{attribute 'no_explicit_call' := 'do not call this function block directly'}
FUNCTION_BLOCK FB_Vector IMPLEMENTS I_Vector, I_Addition, I_Subtraction, I_Multiplication
VAR
	_fX, _fY, _fZ : LREAL;
END_VAR

{attribute 'hide'}
METHOD FB_init : BOOL
VAR_INPUT
	bInitRetains : BOOL; // if TRUE, the retain variables are initialized (warm start / cold start)
	bInCopyCode : BOOL;  // if TRUE, the instance afterwards gets moved into the copy code (online change)
	fX, fY, fZ : LREAL;
END_VAR
THIS^.SetValue(fX, fY, fZ);
END_METHOD

METHOD Minus : I_Subtraction
VAR_INPUT
	ipObject : I_Object;
END_VAR
VAR_OUTPUT
	e : E_OperatorError;
END_VAR
VAR
	ipVector : I_Vector;
END_VAR
Minus := THIS^;

IF NOT __QUERYINTERFACE(ipObject, ipVector) THEN
  e := E_OperatorError.TypeMismatch;
  RETURN;
  END_IF

THIS^._fX := THIS^._fX - ipVector.X;
THIS^._fY := THIS^._fY - ipVector.Y;
THIS^._fZ := THIS^._fZ - ipVector.Z;
END_METHOD

METHOD Plus : I_Addition
VAR_INPUT
	ipObject : I_Object;
END_VAR
VAR_OUTPUT
	e : E_OperatorError;
END_VAR
VAR
	ipVector : I_Vector;
END_VAR
Plus := THIS^;

IF NOT __QUERYINTERFACE(ipObject, ipVector) THEN
  e := E_OperatorError.TypeMismatch; 
  RETURN;
  END_IF

THIS^._fX := THIS^._fX + ipVector.X;
THIS^._fY := THIS^._fY + ipVector.Y;
THIS^._fZ := THIS^._fZ + ipVector.Z;
END_METHOD

METHOD SetValue : REFERENCE TO FB_Vector
VAR_INPUT
	fX, fY, fZ : LREAL;
END_VAR
SetValue REF= THIS^;

THIS^._fX := fX;
THIS^._fY := fY;
THIS^._fZ := fZ;
END_METHOD

METHOD Times : I_Multiplication
VAR_INPUT
	ipObject : I_Object;
END_VAR
VAR_OUTPUT
	e : E_OperatorError;
END_VAR
VAR
	ipNumber : I_Scalar;
	ipVector : I_Vector;
	TmpX, TmpY, TmpZ : LREAL;
END_VAR
Times := THIS^;

// Scale vector.
IF __QUERYINTERFACE(ipObject, ipNumber) THEN 
	THIS^.SetValue( THIS^._fX * ipNumber.ToF64(),
					THIS^._fY * ipNumber.ToF64(),
					THIS^._fZ * ipNumber.ToF64());
	RETURN;
	END_IF

// Do the cross-product.
IF __QUERYINTERFACE(ipObject, ipVector) THEN 
	TmpX := THIS^._fX;
  TmpY := THIS^._fY;
  TmpZ := THIS^._fZ;
  
	THIS^.SetValue(	(TmpY*ipVector.Z) - (TmpZ*ipVector.Y),
					        (TmpZ*ipVector.X) - (TmpX*ipVector.Y),
					        (TmpX*ipVector.Y) - (TmpY*ipVector.X));
	
	RETURN; 
	END_IF

e := E_OperatorError.TypeMismatch;
END_METHOD

METHOD ToArray : ARRAY[0..2] OF LREAL
VAR_INPUT
END_VAR

ToArray[0]:= THIS^._fX;
ToArray[1]:= THIS^._fY;
ToArray[2]:= THIS^._fZ;
END_METHOD

PROPERTY X : LREAL
GET
X := THIS^._fX;
END_GET
SET
THIS^._fX := X;
END_SET
END_PROPERTY

PROPERTY Y : LREAL
GET
Y := THIS^._fY;
END_GET
SET
THIS^._fY:= Y;
END_SET
END_PROPERTY

PROPERTY Z : LREAL
GET
Z := THIS^._fZ;
END_GET
SET
THIS^._fZ := Z;
END_SET
END_PROPERTY

END_FUNCTION_BLOCK

(* stored: Version 1.1.0.1, ProductVersion 3.1.4024.12
   POU FB_Vector: Id {a3e3f989-5383-4684-9365-351b5d5ddbc2}, SpecialFunc None
   Folder Constructor: Id {4d519fb7-d67d-4a3b-ad25-276b7aa36544}
   Folder IOperatorX: Id {dc5b5d9f-5cca-45c6-8635-d968a0da61ca}
   Folder IVector: Id {a72ffef8-55b1-4923-ae3f-21af8125f718}
   Method FB_init: Id {5e146931-1a8b-485c-a8f5-25b63288d0d0}
   Method Minus: Id {8d6c7050-0ff6-4ab0-a242-534401decfff}
   Method Plus: Id {5087b5ff-4e99-4c43-993f-4b57fa3ce74e}
   Method SetValue: Id {d9885a12-06a6-429e-9b7e-42cdf297705b}
   Method Times: Id {d62c470e-1109-45a1-8f8e-9c3f6f9ddf37}
   Method ToArray: Id {426b64b7-c7f6-4e3d-a17e-aee296eec29f}
   Property X: Id {78d98864-2df4-4548-b5b8-7345b73f380f}
   Get Get: Id {c9132885-5c5b-4f0a-b8a2-fcdc7d99b0d7}
   Set Set: Id {1aa968b6-af80-49d0-9736-d65e016dbdaa}
   Property Y: Id {8b210bcc-2877-43dc-bb5c-5e2a0c50e47d}
   Get Get: Id {66ce0378-c4c4-4aa4-830b-5dee598b822e}
   Set Set: Id {8e499bf2-af60-4e77-a1aa-4e3f0f629d69}
   Property Z: Id {fb0365b7-1fdd-4a89-828a-5fa742effd17}
   Get Get: Id {29e3d436-10f6-4404-a55f-a061213ae47a}
   Set Set: Id {a36fee45-ea70-4a11-8ec2-87c5e753b9b6} *)
